FUNCTION Control24V
VAR_INPUT
END_VAR
VAR
	fbTon : TON;
END_VAR

//Control 24V for simulation
//This is the simulation of the safety circuit. Power supply for the output modules.
IF (MeasuringData.ES1NC AND MeasuringData.ES2NC AND Inputs.Control24VButton) THEN
	fbTon(IN := TRUE, PT := T#3S);
ELSE
	fbTon(IN := FALSE);
END_IF

MeasuringData.ControlSupplyOK := fbTon.Q;

END_FUNCTION

(* stored: Version 1.1.0.1, ProductVersion 3.1.4024.13
   POU Control24V: Id {454e5c67-702f-480f-863a-dbbb804afe59}, SpecialFunc None *)
